{attribute 'qualified_only'}
VAR_GLOBAL
		EtherCAT_Master_EPxxxx : EtherCAT_Master_EPxxxx_2B438D5B;
END_VAR

(* stored: Version 1.2.0.0, ProductVersion 3.1.4024.9
   GVL GVL_iXlinker: Id {7d35b76d-e9ca-449f-acc5-5f1840e79e63} *)
